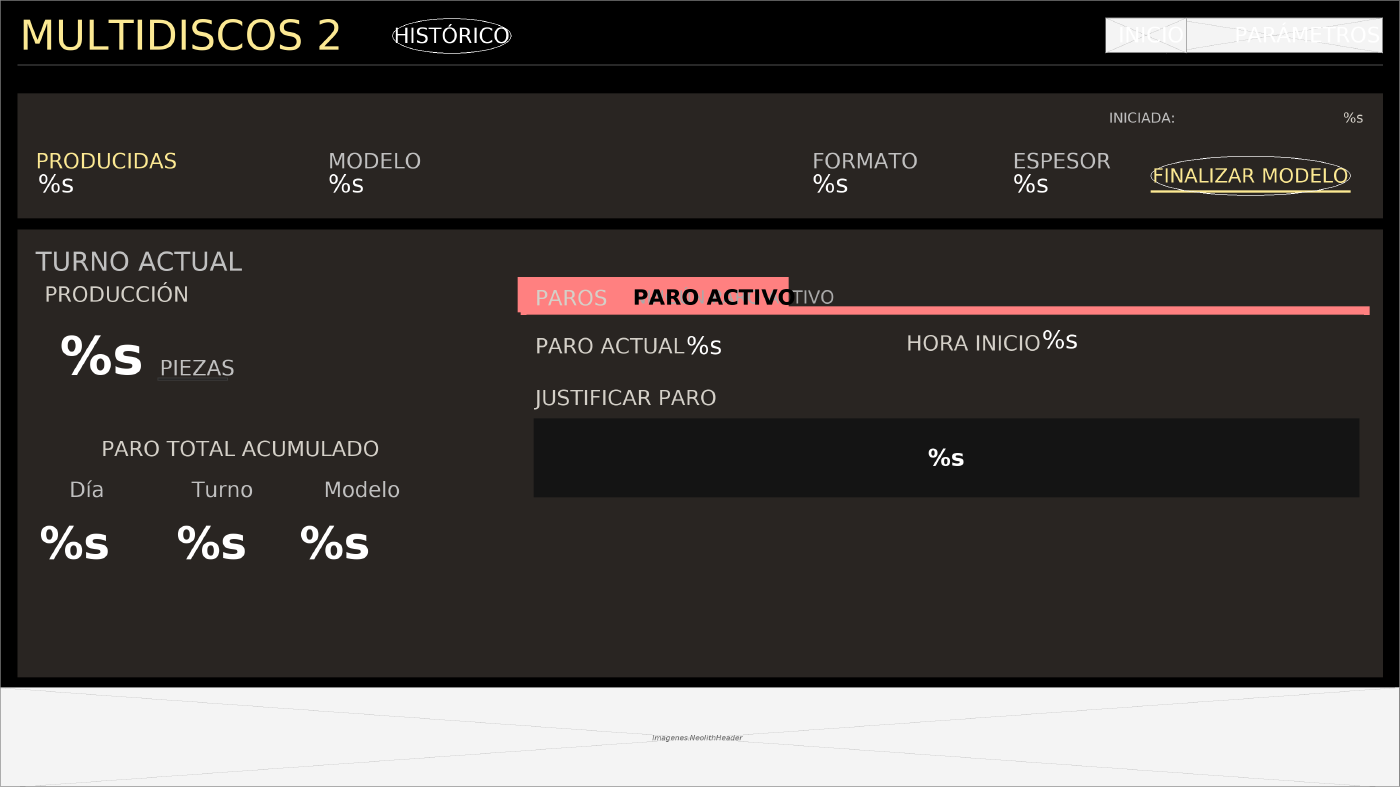
VISUALIZATION Home_Multidis2  // 1920x1080
    Ellipse (1479,1885 456x77), "Fin de producción del modelo"
        OnMouseClick: OpenDialog Dialog=V_Emerg_Fin_Prod_Md2, OpenModal=True, OpenCentered=True
    Lamp1 (869,1190 94x97), variable: FuncParoNodoMultidiscos.Funci_Multidiscos2.Fotocelula, style: Lamp-Lamp1-Yellow
    Rectangle (994,1445 183x30), "%s", text variable: FuncParoNodoCorteH4Remote1.Funci_CortHum4.H_InParo_Ftc, invisible if: FuncParoNodoMultidiscos.Funci_Multidiscos2.M_SinParo_Ftc
    Label (758,1444 239x30), "Hora Inicio del paro", invisible if: FuncParoNodoMultidiscos.Funci_Multidiscos2.M_SinParo_Ftc
    Rectangle (994,1503 192x30), "%s", text variable: FuncParoNodoCorteH4Remote1.Funci_CortHum4.Min_Parado_Ftc, invisible if: FuncParoNodoMultidiscos.Funci_Multidiscos2.M_SinParo_Ftc
    Label (793,1503 204x30), "Minutos Parado", invisible if: FuncParoNodoMultidiscos.Funci_Multidiscos2.M_SinParo_Ftc
    Label (753,1558 244x30), "Tiempo entre Piezas"
    Label (742,1594 255x62), "Tiempo entre Piezas Anterior"
    Rectangle (172,1318 183x123), "%s", text variable: FuncParoNodoMultidiscos.Funci_Multidiscos2.Cont_Piezas_Ftc
    Rectangle (994,1558 192x30), "%s", text variable: FuncParoNodoCorteH4Remote1.Funci_CortHum4.t_Entre_Piez_Ftc
    Rectangle (994,1610 192x30), "%s", text variable: FuncParoNodoCorteH4Remote1.Funci_CortHum4.t_Entr_Piez_Ante_Ftc
    Label (718,1127 397x30), "Sensor presencia tabla"
    Label (753,1348 326x30), "En producción todo OK", invisible if: FuncParoNodoMultidiscos.Funci_Multidiscos2.MParo_Ftc
    Label (571,1279 235x59), "Línea en paro", invisible if: FuncParoNodoMultidiscos.Funci_Multidiscos2.M_SinParo_Ftc
    Label (85,1180 361x144), "Número de losas"
    Label (1390,1230 361x56), "Modelo actual"
    Rectangle (1235,1324 671x53), "%s", text variable: FuncParoNodoMultidiscos.sModeloActualTabla_MD2
    Label (1390,1615 361x56), "Espesor"
    Rectangle (1235,1704 671x53), "%s", text variable: FuncParoNodoMultidiscos.sEspesorActualTabla_MD2
    Label (1390,1417 361x56), "Formato"
    Rectangle (1235,1506 671x53), "%s", text variable: FuncParoNodoMultidiscos.sFormatoActualTabla_MD2
    Rectangle (1533,1124 300x30), "%s", text variable: FuncParoNodoMultidiscos.sFechaInicModeloTab_MD2
    Label (1178,1125 354x30), "Fecha inicio del modelo actual"
    Rectangle (56,1801 1380x154), "%s", text variable: FuncParoNodoMultidiscos.Funci_Multidiscos2.S_Justi_Paro_Ftc, invisible if: FuncParoNodoMultidiscos.Funci_Multidiscos2.M_SinParo_Ftc
        OnMouseDown: write the text variable via Edit
    Label (55,1710 1381x106), "JUSTIFICAR EL PARO ACTUAL", invisible if: FuncParoNodoCorteH4Remote1.Funci_CortHum4.M_SinParo_Ftc
    Rectangle (24,315 1872x614)
    Rectangle (24,128 1872x171)
    Rectangle (24,88 1872x2)
    Label (24,16 514x64), "MULTIDISCOS 2"
    Rectangle (1426,451 183x30), "%s", text variable: FuncParoNodoCorteH4Remote1.Funci_CortHum4.H_InParo_Ftc, invisible if: FuncParoNodoMultidiscos.Funci_Multidiscos2.M_SinParo_Ftc
    Rectangle (938,459 192x30), "%s", text variable: FuncParoNodoCorteH4Remote1.Funci_CortHum4.Min_Parado_Ftc, invisible if: FuncParoNodoMultidiscos.Funci_Multidiscos2.M_SinParo_Ftc
    Rectangle (1573,147 300x30), "%s", text variable: FuncParoNodoMultidiscos.sFechaInicModeloTab_MD2
    Label (1518,147 99x30), "INICIADA:"
    Rectangle (732,574 1132x108), "%s", text variable: FuncParoNodoMultidiscos.Funci_Multidiscos2.S_Justi_Paro_Ftc, invisible if: FuncParoNodoMultidiscos.Funci_Multidiscos2.M_SinParo_Ftc
        OnMouseDown: write the text variable via Edit
    Image (1600,24 296x48), "PARÁMETROS"
        OnMouseClick: change screen: Ajustes_Multidiscos2
    Image (1516,24 111x48), "INICIO"
        OnMouseClick: change screen: Home_Sel_Maq
    Rectangle (447,232 671x40), "%s", text variable: FuncParoNodoMultidiscos.sModeloActualTabla_MD2
    Rectangle (1386,232 120x40), "%s", text variable: FuncParoNodoMultidiscos.sEspesorActualTabla_MD2
    Rectangle (1111,232 321x40), "%s", text variable: FuncParoNodoMultidiscos.sFormatoActualTabla_MD2
    Label (447,203 487x36), "MODELO"
    Label (1111,203 156x36), "FORMATO"
    Label (1386,203 156x36), "ESPESOR"
    Label (46,203 199x36), "PRODUCIDAS"
    Rectangle (49,232 248x40), "%s", text variable: FuncParoNodoCorteH4Remote1.sEspesorActualTabla
    Group (1578,214 274x54)
        Rectangle (0,47 274x3)
        Ellipse (0,0 274x54), "FINALIZAR MODELO"
            OnMouseClick: OpenDialog Dialog=V_Emerg_Fin_Prod_Md2, OpenModal=True, OpenCentered=True
    Label (46,332 390x54), "TURNO ACTUAL"
    Label (58,386 199x36), "PRODUCCIÓN"
    Label (731,457 261x36), "PARO ACTUAL", invisible if: FuncParoNodoMultidiscos.Funci_Multidiscos2.M_SinParo_Ftc
    Label (1240,453 261x36), "HORA INICIO", invisible if: FuncParoNodoMultidiscos.Funci_Multidiscos2.M_SinParo_Ftc
    Rectangle (79,444 183x88), "%s", text variable: FuncParoNodoMultidiscos.Funci_Multidiscos2.Cont_Piezas_Ftc
    Label (216,487 106x36), "PIEZAS"
    Rectangle (216,518 96x4), colour toggle: FuncParoNodoCorteH4Remote1.Funci_CortHum4.Fotocelula
    Label (731,528 261x36), "JUSTIFICAR PARO", invisible if: FuncParoNodoMultidiscos.Funci_Multidiscos2.M_SinParo_Ftc
    Rectangle (714,424 1164x4), invisible if: FuncParoNodoMultidiscos.Funci_Multidiscos2.M_SinParo_Ftc
    Rectangle (710,380 371x48), invisible if: FuncParoNodoMultidiscos.Funci_Multidiscos2.M_SinParo_Ftc
    Label (731,391 199x36), "PAROS"
    Label (865,393 326x30), "NINGÚN PARO ACTIVO", invisible if: FuncParoNodoMultidiscos.Funci_Multidiscos2.MParo_Ftc
    Label (865,393 235x30), "PARO ACTIVO", invisible if: FuncParoNodoMultidiscos.Funci_Multidiscos2.M_SinParo_Ftc
    Ellipse (538,25 163x48), "HISTÓRICO"
        OnMouseClick: change screen: HistTablaTablas_Ch4
    Image (-7,943 1927x139), image: Imagenes.NeolithHeader
    Label (136,598 367x36), "PARO TOTAL ACUMULADO"
    Rectangle (51,701 183x88), "%s", text variable: FuncParoNodoMultidiscos.Funci_Multidiscos2.fbTiempParoAcumDiario.t_Acumulado
    Label (92,654 76x36), "Día"
    Rectangle (239,701 167x88), "%s", text variable: FuncParoNodoMultidiscos.Funci_Multidiscos2.fbTiempParoAcumTurno.t_Acumulado
    Label (260,654 102x36), "Turno"
    Rectangle (408,701 183x88), "%s", text variable: FuncParoNodoMultidiscos.Funci_Multidiscos2.fbTiempParoAcumModelo.t_Acumulado
    Label (441,654 118x36), "Modelo"
END_VISUALIZATION

(* stored: Version 1.1.0.1, ProductVersion 3.1.4024.12
   Visu Home_Multidis2: Id {dffd5fcd-21e9-460b-bbb5-641c7dfc56fe} *)
